Staubli VAL3: main.pgx

public program main()
  local num i
  local bool l_bSave
  local string sButton[3]
  local string sItems[2]
begin
  call onStart()
  do
    call refresh()
    nKey=getKey()
    call use:listevent(nKey,nIndex,sEvent)
    nView=use:nView
    nSelected=nIndex
    //
    // OVERRIDE NORMAL FUNCTIONALITY-> POLYMORPHISM
    //
    switch nKey
      case 264
        // left
        call onLeftEvent()
      break
      case 268
        // right
        call onRightEvent()
      break
      case 271
        // test
        call onF1Event()
      break
      case 272
        //
        call onF2Event()
      break
      case 273
        call onF3Event()
      break
      case 274
        call onF4Event()
      break
      case 275
        //
        call onF5Event()
      break
      case 276
        // set type
        call onF6Event()
      break
      case 277
        // DELETE
        call onF7Event()
      break
      case 278
        // NEW
        call onF8Event()
        l_bSave=true
      break
      case 270
        call onEnterEvent()
      break
    endSwitch
    // release the resource
    delay(0)
  until nKey==255 and isKeyPressed(289)==false
  // exit
  call onExit(l_bSave)
end
